{attribute 'qualified_only'}
{attribute 'strict'}
{attribute 'to_string'}
TYPE E_MarkMode :
(
	AutoDefault := 0,       // a start mark and all intermediate marks, given by formula
	None        := 1,        // no marks defined, simulate marks
	OneDefault  := 2,       // only one "default* mark at beginning of sheet
  OneTriangle := 3       // only one "old" mark with a rectancular triangle
) UINT := AutoDefault ;
END_TYPE

(* stored: Version 1.1.0.1, ProductVersion 3.1.4024.11
   EnumerationTextList E_MarkMode: Id {f985e454-5689-4383-95f3-db9fa8e3dcf3} *)
